SUBAPPLICATION Uebung_002_AX (* DigitalInput_I1 auf DigitalOutput_Q1/_Q2, mit Plug and Socket *)
  (* Standard: 61499-2; Description: Copyright (c) 2023 Meisterschulen am Ostbahnhof This program and the accompanying materials are made available under the terms of the Eclipse Public License 2.0 which is available at https://www.eclipse.org/legal/epl-2.0/ SPDX-License-Identifier: EPL-2.0 *)
  (* Version 1.0, 2023-10-23, Franz Höpfinger, Meisterschulen am Ostbahnhof *)
  IMPORT logiBUS::io::DI::logiBUS_DI::Input_I1;
  IMPORT logiBUS::io::DQ::logiBUS_DO::Output_Q1;
  IMPORT logiBUS::io::DQ::logiBUS_DO::Output_Q2;
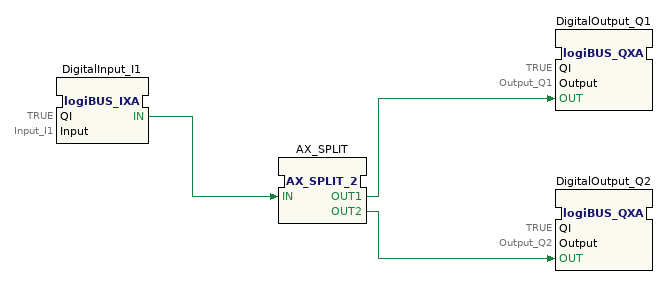
  FBS
    DigitalInput_I1 : logiBUS::io::DI::logiBUS_IXA(QI := TRUE, Input := Input_I1);
    DigitalOutput_Q1 : logiBUS::io::DQ::logiBUS_QXA(QI := TRUE, Output := Output_Q1);
    DigitalOutput_Q2 : logiBUS::io::DQ::logiBUS_QXA(QI := TRUE, Output := Output_Q2);
    AX_SPLIT : adapter::events::unidirectional::AX_SPLIT_2;
  END_FBS
  ADAPTER_CONNECTIONS
    DigitalInput_I1.IN TO AX_SPLIT.IN;
    AX_SPLIT.OUT1 TO DigitalOutput_Q1.OUT;
    AX_SPLIT.OUT2 TO DigitalOutput_Q2.OUT;
  END_CONNECTIONS
END_SUBAPPLICATION
